// TIA Portal project "LAB3Simu" (V18)

(* hardware
DEVICE "S7-1500/ET200MP station_1"  S7-1500 station
   slot 0: "Rail_0"  Rack  6ES7 590-1***0-0AA0
   slot 1: "PLC_1"  CPU 1511-1 PN  6ES7 511-1AK00-0AB0  V1.8
      slot 3: "CPU display_1"  6ES7591-1AA00-0AA0
      slot 32768: "PROFINET interface_1"  X1
         slot 32769: "Port_1"  X1 P1
         slot 32770: "Port_2"  X1 P2
   slot 2: "CM 1542-5_1"  CM 1542-5  6GK7 542-5DX00-0XE0  V1.0
   slot 3: "DI 16x24VDC HF_1"  DI 16x24VDC HF  6ES7 521-1BH00-0AB0  V1.0
   slot 4: "DQ 16x24VDC/0.5A ST_1"  DQ 16x24VDC/0.5A ST  6ES7 522-1BH00-0AB0  V1.0
   slot 5: "AI 8xU/I/RTD/TC ST_1"  AI 8xU/I/RTD/TC ST  6ES7 531-7KF00-0AB0  V1.0
   slot 6: "AQ 4xU/I ST_1"  AQ 4xU/I ST  6ES7 532-5HD00-0AB0  V1.0
DEVICE "HMI_1"  KP700 Comfort
   slot 0: "HMI_1"  KP700 Comfort  6AV2 124-1GC01-0AX0  17.0.0.0
   slot 1: "HMI_RT_1"  KP700 Comfort  6AV2 124-1GC01-0AX0  17.0.0.0
   slot 5: "HMI_1.IE_CP_1"  PROFINET Interface  17.0.0.0
      slot 1: "PROFINET Interface_1"  PROFINET Interface
         slot 1: "Port_1"  Port
         slot 2: "Port_2"  Port
   slot 7: "HMI_1.MPI/DP_CP_1"  MPI/DP Interface  17.0.0.0
*)

// ===== PLC "PLC_1"  CPU 1511-1 PN =====

VAR_GLOBAL   // PLC tag table "Default tag table"
   "Btn_Ciclo_INIT" AT %M0.0 : Bool;
   "Btn_Ciclo_Cont" AT %M0.1 : Bool;
   "Btn_Parada" AT %M0.2 : Bool;
   "Btn_Emergencia" AT %M0.3 : Bool;
   "Sens_PP" AT %M0.4 : Bool;
   "Sens_PC" AT %M0.5 : Bool;
   "Sens_SM" AT %M0.6 : Bool;
   "A0" AT %M0.7 : Bool;
   "B0" AT %M1.0 : Bool;
   "C0" AT %M1.1 : Bool;
   "D0" AT %M1.2 : Bool;
   "E0" AT %M1.3 : Bool;
   "F0" AT %M1.4 : Bool;
   "A1" AT %M1.5 : Bool;
   "B1" AT %M1.6 : Bool;
   "C1" AT %M1.7 : Bool;
   "D1" AT %M2.0 : Bool;
   "E1" AT %M2.1 : Bool;
   "F1" AT %M2.2 : Bool;
   "Cil_A_+" AT %M2.3 : Bool;
   "Cil_A_-" AT %M2.4 : Bool;
   "Cil_B_Out" AT %M2.5 : Bool;
   "Cil_C_Out" AT %M2.6 : Bool;
   "Cil_D_Out" AT %M2.7 : Bool;
   "Cil_E_+" AT %M3.0 : Bool;
   "Cil_E_-" AT %M3.1 : Bool;
   "Cil_F_+" AT %M3.2 : Bool;
   "Cil_F_-" AT %M3.3 : Bool;
   "Alarma_Stock" AT %M3.4 : Bool;
   "Marca_D_OK" AT %M3.5 : Bool;
   "reset" AT %M3.6 : Bool;
   "start" AT %M3.7 : Bool;
   "stop" AT %M4.0 : Bool;
   "PE" AT %M4.1 : Bool;
   "ALM_start" AT %M4.2 : Bool;
   "ALM_stop" AT %M4.3 : Bool;
   "ALM_em" AT %M4.4 : Bool;
   "block_start" AT %M4.5 : Bool;
   "Alarma_pp" AT %M4.6 : Bool;
   "Alarma_pc" AT %M4.7 : Bool;
   "Marca_start" AT %M5.0 : Bool;
END_VAR

DATA_BLOCK "GRAFCET_DB"   // DB2
{ S7_Optimized_Access := 'TRUE' }
VERSION : 0.1
// stored: InstanceOfName GRAFCET
"GRAFCET"
BEGIN
END_DATA_BLOCK

DATA_BLOCK "FUB_DB"   // DB3
{ S7_Optimized_Access := 'TRUE' }
VERSION : 0.1
// stored: InstanceOfName FUB
"FUB"
BEGIN
END_DATA_BLOCK

DATA_BLOCK "AWL_DB"   // DB4
{ S7_Optimized_Access := 'TRUE' }
VERSION : 0.1
// stored: InstanceOfName AWL
"AWL"
BEGIN
END_DATA_BLOCK

// folder: System blocks/Program resources

DATA_BLOCK "IEC_Timer_0_DB"   // DB1
{ S7_Optimized_Access := 'TRUE' }
AUTHOR : Simatic
FAMILY : IEC
NAME : IEC_TMR
VERSION : 1.0
// stored: InstanceOfName IEC_TIMER
"IEC_TIMER"
BEGIN
END_DATA_BLOCK

// folder: (top level)

FUNCTION_BLOCK "GRAFCET"   // FB1, GRAPH_PLUS
{ S7_Optimized_Access := 'TRUE' }
VERSION : 0.1
   VAR_INPUT
      OFF_SQ : Bool := false;   // Turn sequence off
      INIT_SQ : Bool := false;   // Set sequence to initial state
      ACK_EF : Bool := false;   // Acknowledge all errors and faults
      S_PREV : Bool := false;   // Output previous step in parameter S_NO
      S_NEXT : Bool := false;   // Indicate next step in parameter S_NO
      SW_AUTO : Bool := false;   // Automatic mode
      SW_TAP : Bool := false;   // Semiautomatic/switch with transition
      SW_TOP : Bool := false;   // Semiautomatic/ignore transition
      SW_MAN : Bool := false;   // Manual mode
      S_SEL : Int := 0;   // Select step to be output to S_NO
      S_ON : Bool := false;   // Activate step indicated in S_NO
      S_OFF : Bool := false;   // Disable step indicated in S_NO
      T_PUSH : Bool := false;   // Enable transition to switch in semi automatic mode
   END_VAR
   VAR_OUTPUT
      S_NO : Int := 0;   // Step number
      S_MORE : Bool := false;   // More steps are available and can be shown in S_NO
      S_ACTIVE : Bool := false;   // Step indicated in S_NO is active
      ERR_FLT : Bool := false;   // Interlock or supervision group error
      AUTO_ON : Bool := false;   // Automatic mode is active
      TAP_ON : Bool := false;   // Semiautomatic mode/step with transition enabled
      TOP_ON : Bool := false;   // Semiautomatic mode/ignore transition enabled
      MAN_ON : Bool := false;   // Manual mode is active
   END_VAR
   VAR
      HMI_INFO : Array[0..8] of UInt;
      IF_PAR : G7_IfParPlus_V2;
      RT_DATA : G7_RTDataPlus_V2;   // Internal data area
      Trans1 : G7_TransitionPlus_V2;   // Transition structure
      Trans2 : G7_TransitionPlus_V2;   // Transition structure
      Trans3 : G7_TransitionPlus_V2;   // Transition structure
      Trans4 : G7_TransitionPlus_V2;   // Transition structure
      Trans5 : G7_TransitionPlus_V2;   // Transition structure
      Trans6 : G7_TransitionPlus_V2;   // Transition structure
      Trans7 : G7_TransitionPlus_V2;   // Transition structure
      Trans8 : G7_TransitionPlus_V2;   // Transition structure
      Trans9 : G7_TransitionPlus_V2;   // Transition structure
      Trans10 : G7_TransitionPlus_V2;   // Transition structure
      Trans11 : G7_TransitionPlus_V2;   // Transition structure
      Trans12 : G7_TransitionPlus_V2;   // Transition structure
      Trans13 : G7_TransitionPlus_V2;   // Transition structure
      Trans14 : G7_TransitionPlus_V2;   // Transition structure
      Trans15 : G7_TransitionPlus_V2;   // Transition structure
      Trans16 : G7_TransitionPlus_V2;   // Transition structure
      Trans17 : G7_TransitionPlus_V2;   // Transition structure
      Trans18 : G7_TransitionPlus_V2;   // Transition structure
      Trans19 : G7_TransitionPlus_V2;   // Transition structure
      Trans20 : G7_TransitionPlus_V2;   // Transition structure
      Trans21 : G7_TransitionPlus_V2;   // Transition structure
      Trans22 : G7_TransitionPlus_V2;   // Transition structure
      Trans23 : G7_TransitionPlus_V2;   // Transition structure
      "Reset/Reposo" : G7_StepPlus_V2;   // Step structure
      "A+" : G7_StepPlus_V2;   // Step structure
      "A-" : G7_StepPlus_V2;   // Step structure
      "B+" : G7_StepPlus_V2;   // Step structure
      "C+" : G7_StepPlus_V2;   // Step structure
      "B-" : G7_StepPlus_V2;   // Step structure
      "D sale" : G7_StepPlus_V2;   // Step structure
      "D-" : G7_StepPlus_V2;   // Step structure
      "C-" : G7_StepPlus_V2;   // Step structure
      "E+,F+" : G7_StepPlus_V2;   // Step structure
      "E-,F-" : G7_StepPlus_V2;   // Step structure
      "A++" : G7_StepPlus_V2;   // Step structure
      "A--" : G7_StepPlus_V2;   // Step structure
      "B++" : G7_StepPlus_V2;   // Step structure
      "C++" : G7_StepPlus_V2;   // Step structure
      "B--" : G7_StepPlus_V2;   // Step structure
      D_out : G7_StepPlus_V2;   // Step structure
      "D++" : G7_StepPlus_V2;   // Step structure
      "D--" : G7_StepPlus_V2;   // Step structure
      "E,F++" : G7_StepPlus_V2;   // Step structure
      "E,F--" : G7_StepPlus_V2;   // Step structure
      "Cilindros -" : G7_StepPlus_V2;   // Step structure
      SINI : Array[0..1] of USInt;
      LSTT : Array[0..22] of USInt;
      ATAJ : Array[0..22] of USInt;
      ATAB : Array[0..22] of USInt;
      PSTT : Array[0..22] of USInt;
      NSTT : Array[0..22] of USInt;
      ASSJ : Array[0..21] of USInt;
      ASSB : Array[0..21] of USInt;
      PTTS : Array[0..21] of USInt;
      NTTS : Array[0..21] of USInt;
      SW_SQTS : Array[0..21] of USInt;
      SWITCH : Array[0..1] of USInt;
      TVX : Array[0..3] of USInt;
      TTX : Array[0..3] of USInt;
      TSX : Array[0..1] of USInt;
      S00X : Array[0..1] of USInt;
      SOFFX : Array[0..1] of USInt;
      SONX : Array[0..1] of USInt;
      SAX : Array[0..1] of USInt;
      SERRX : Array[0..22] of USInt;
      SMX : Array[0..22] of USInt;
      S0X : Array[0..22] of USInt;
      S1X : Array[0..22] of USInt;
      IL_ALARM_INST : Program_Alarm;
      SUP_ALARM_INST : Program_Alarm;
      STEP_TIME_ALARM_INST : Program_Alarm;
      IEC_TIMER_INST : IEC_TIMER;
      TRANSACTION_FLAG : Bool := false;
   END_VAR
   // SINI[0] := 2;
   // LSTT[0] := 255;
   // LSTT[1] := 255;
   // LSTT[2] := 255;
   // LSTT[3] := 255;
   // LSTT[4] := 255;
   // LSTT[5] := 255;
   // LSTT[6] := 255;
   // LSTT[7] := 255;
   // LSTT[8] := 255;
   // LSTT[9] := 255;
   // LSTT[10] := 255;
   // LSTT[11] := 255;
   // LSTT[12] := 255;
   // LSTT[13] := 255;
   // LSTT[14] := 255;
   // LSTT[15] := 255;
   // LSTT[16] := 255;
   // LSTT[17] := 255;
   // LSTT[18] := 255;
   // LSTT[19] := 255;
   // LSTT[20] := 255;
   // ATAJ[1] := 1;
   // ATAJ[2] := 2;
   // ATAJ[3] := 3;
   // ATAJ[4] := 4;
   // ATAJ[5] := 5;
   // ATAJ[6] := 6;
   // ATAJ[7] := 7;
   // ATAJ[8] := 8;
   // ATAJ[9] := 9;
   // ATAJ[10] := 10;
   // ATAJ[11] := 11;
   // ATAJ[12] := 12;
   // ATAJ[13] := 13;
   // ATAJ[14] := 14;
   // ATAJ[15] := 15;
   // ATAJ[16] := 16;
   // ATAJ[17] := 17;
   // ATAJ[18] := 18;
   // ATAJ[19] := 19;
   // ATAJ[20] := 20;
   // ATAJ[21] := 21;
   // ATAB[0] := 11;
   // ATAB[1] := 1;
   // ATAB[2] := 2;
   // ATAB[3] := 3;
   // ATAB[4] := 4;
   // ATAB[5] := 5;
   // ATAB[6] := 6;
   // ATAB[7] := 7;
   // ATAB[8] := 8;
   // ATAB[9] := 9;
   // ATAB[10] := 10;
   // ATAB[12] := 12;
   // ATAB[13] := 13;
   // ATAB[14] := 14;
   // ATAB[15] := 15;
   // ATAB[16] := 16;
   // ATAB[17] := 17;
   // ATAB[18] := 18;
   // ATAB[19] := 19;
   // ATAB[20] := 20;
   // ATAB[21] := 21;
   // PSTT[1] := 1;
   // PSTT[2] := 2;
   // PSTT[3] := 3;
   // PSTT[4] := 4;
   // PSTT[5] := 5;
   // PSTT[6] := 6;
   // PSTT[7] := 7;
   // PSTT[8] := 8;
   // PSTT[9] := 9;
   // PSTT[10] := 10;
   // PSTT[12] := 11;
   // PSTT[13] := 12;
   // PSTT[14] := 13;
   // PSTT[15] := 14;
   // PSTT[16] := 15;
   // PSTT[17] := 16;
   // PSTT[18] := 17;
   // PSTT[19] := 18;
   // PSTT[20] := 19;
   // PSTT[21] := 20;
   // NSTT[0] := 1;
   // NSTT[1] := 2;
   // NSTT[2] := 3;
   // NSTT[3] := 4;
   // NSTT[4] := 5;
   // NSTT[5] := 6;
   // NSTT[6] := 7;
   // NSTT[7] := 8;
   // NSTT[8] := 9;
   // NSTT[9] := 10;
   // NSTT[10] := 255;
   // NSTT[11] := 11;
   // NSTT[12] := 12;
   // NSTT[13] := 13;
   // NSTT[14] := 14;
   // NSTT[15] := 15;
   // NSTT[16] := 16;
   // NSTT[17] := 17;
   // NSTT[18] := 18;
   // NSTT[19] := 19;
   // NSTT[20] := 20;
   // ASSJ[1] := 1;
   // ASSJ[2] := 2;
   // ASSJ[3] := 3;
   // ASSJ[4] := 4;
   // ASSJ[5] := 5;
   // ASSJ[6] := 6;
   // ASSJ[7] := 7;
   // ASSJ[8] := 8;
   // ASSJ[9] := 9;
   // ASSJ[10] := 10;
   // ASSJ[11] := 11;
   // ASSJ[12] := 12;
   // ASSJ[13] := 13;
   // ASSJ[14] := 14;
   // ASSJ[15] := 15;
   // ASSJ[16] := 16;
   // ASSJ[17] := 17;
   // ASSJ[18] := 18;
   // ASSJ[19] := 19;
   // ASSJ[20] := 20;
   // ASSB[1] := 1;
   // ASSB[2] := 2;
   // ASSB[3] := 3;
   // ASSB[4] := 4;
   // ASSB[5] := 5;
   // ASSB[6] := 6;
   // ASSB[7] := 7;
   // ASSB[8] := 8;
   // ASSB[9] := 9;
   // ASSB[10] := 10;
   // ASSB[11] := 11;
   // ASSB[12] := 12;
   // ASSB[13] := 13;
   // ASSB[14] := 14;
   // ASSB[15] := 15;
   // ASSB[16] := 16;
   // ASSB[17] := 17;
   // ASSB[18] := 18;
   // ASSB[19] := 19;
   // ASSB[20] := 20;
   // PTTS[0] := 255;
   // PTTS[2] := 1;
   // PTTS[3] := 2;
   // PTTS[4] := 3;
   // PTTS[5] := 4;
   // PTTS[6] := 5;
   // PTTS[7] := 6;
   // PTTS[8] := 7;
   // PTTS[9] := 8;
   // PTTS[10] := 9;
   // PTTS[11] := 11;
   // PTTS[12] := 12;
   // PTTS[13] := 13;
   // PTTS[14] := 14;
   // PTTS[15] := 15;
   // PTTS[16] := 16;
   // PTTS[17] := 17;
   // PTTS[18] := 18;
   // PTTS[19] := 19;
   // PTTS[20] := 20;
   // NTTS[1] := 1;
   // NTTS[2] := 2;
   // NTTS[3] := 3;
   // NTTS[4] := 4;
   // NTTS[5] := 5;
   // NTTS[6] := 6;
   // NTTS[7] := 7;
   // NTTS[8] := 8;
   // NTTS[9] := 9;
   // NTTS[10] := 10;
   // NTTS[11] := 12;
   // NTTS[12] := 13;
   // NTTS[13] := 14;
   // NTTS[14] := 15;
   // NTTS[15] := 16;
   // NTTS[16] := 17;
   // NTTS[17] := 18;
   // NTTS[18] := 19;
   // NTTS[19] := 20;
   // NTTS[20] := 21;
   // SW_SQTS[1] := 1;
   // SW_SQTS[2] := 1;
   // SW_SQTS[3] := 1;
   // SW_SQTS[4] := 1;
   // SW_SQTS[5] := 1;
   // SW_SQTS[6] := 1;
   // SW_SQTS[7] := 1;
   // SW_SQTS[8] := 1;
   // SW_SQTS[9] := 1;
   // SW_SQTS[10] := 1;
   // SW_SQTS[11] := 2;
   // SW_SQTS[12] := 2;
   // SW_SQTS[13] := 2;
   // SW_SQTS[14] := 2;
   // SW_SQTS[15] := 2;
   // SW_SQTS[16] := 2;
   // SW_SQTS[17] := 2;
   // SW_SQTS[18] := 2;
   // SW_SQTS[19] := 2;
   // SW_SQTS[20] := 2;
   // TVX[0] := 16#1;
   // TTX[0] := 16#1;
   // TSX[0] := 16#1;
   // S00X[0] := 16#1;
   // SOFFX[0] := 16#1;
   // SONX[0] := 16#1;
   // SAX[0] := 16#1;
   // SERRX[0] := 16#1;
   // SMX[0] := 16#1;
   // S0X[0] := 16#1;
   // S1X[0] := 16#1;
   // LSTT[22] := 255;
   // ATAJ[22] := 22;
   // ATAB[22] := 22;
   // PSTT[0] := 21;
   // PSTT[11] := 21;
   // NSTT[22] := 21;
   // ASSJ[21] := 21;
   // ASSB[21] := 21;
   // PTTS[21] := 22;
   // NTTS[0] := 22;
BEGIN
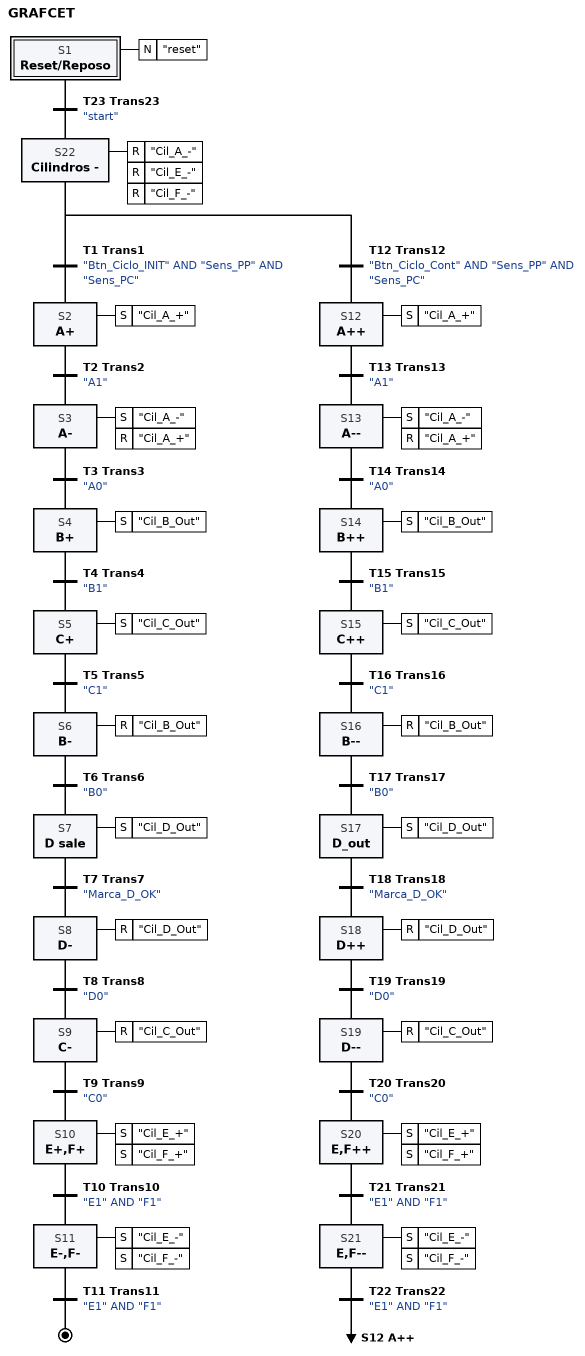
   // sequencer 1
   INITIAL_STEP "Reset/Reposo":   // S1, max time T#10S, warning time T#7S
              N    "reset"
   END_STEP
   TRANSITION Trans23 FROM "Reset/Reposo" TO "Cilindros -"   // T23
      := "start";
   END_TRANSITION
   STEP "A+":   // S2, max time T#10S, warning time T#7S
              S    "Cil_A_+"
   END_STEP
   TRANSITION Trans2 FROM "A+" TO "A-"   // T2
      := "A1";
   END_TRANSITION
   STEP "A-":   // S3, max time T#10S, warning time T#7S
              S    "Cil_A_-"
              R    "Cil_A_+"
   END_STEP
   TRANSITION Trans3 FROM "A-" TO "B+"   // T3
      := "A0";
   END_TRANSITION
   STEP "B+":   // S4, max time T#10S, warning time T#7S
              S    "Cil_B_Out"
   END_STEP
   TRANSITION Trans4 FROM "B+" TO "C+"   // T4
      := "B1";
   END_TRANSITION
   STEP "C+":   // S5, max time T#10S, warning time T#7S
              S    "Cil_C_Out"
   END_STEP
   TRANSITION Trans5 FROM "C+" TO "B-"   // T5
      := "C1";
   END_TRANSITION
   STEP "B-":   // S6, max time T#10S, warning time T#7S
              R    "Cil_B_Out"
   END_STEP
   TRANSITION Trans6 FROM "B-" TO "D sale"   // T6
      := "B0";
   END_TRANSITION
   STEP "D sale":   // S7, max time T#10S, warning time T#7S
              S    "Cil_D_Out"
   END_STEP
   TRANSITION Trans7 FROM "D sale" TO "D-"   // T7
      := "Marca_D_OK";
   END_TRANSITION
   STEP "D-":   // S8, max time T#10S, warning time T#7S
              R    "Cil_D_Out"
   END_STEP
   TRANSITION Trans8 FROM "D-" TO "C-"   // T8
      := "D0";
   END_TRANSITION
   STEP "C-":   // S9, max time T#10S, warning time T#7S
              R    "Cil_C_Out"
   END_STEP
   TRANSITION Trans9 FROM "C-" TO "E+,F+"   // T9
      := "C0";
   END_TRANSITION
   STEP "E+,F+":   // S10, max time T#10S, warning time T#7S
              S    "Cil_E_+"
              S    "Cil_F_+"
   END_STEP
   TRANSITION Trans10 FROM "E+,F+" TO "E-,F-"   // T10
      := "E1" AND "F1";
   END_TRANSITION
   STEP "E-,F-":   // S11, max time T#10S, warning time T#7S
              S    "Cil_E_-"
              S    "Cil_F_-"
   END_STEP
   TRANSITION Trans11 FROM "E-,F-" TO END   // T11
      := "E1" AND "F1";
   END_TRANSITION
   STEP "A++":   // S12, max time T#10S, warning time T#7S
              S    "Cil_A_+"
   END_STEP
   TRANSITION Trans13 FROM "A++" TO "A--"   // T13
      := "A1";
   END_TRANSITION
   STEP "A--":   // S13, max time T#10S, warning time T#7S
              S    "Cil_A_-"
              R    "Cil_A_+"
   END_STEP
   TRANSITION Trans14 FROM "A--" TO "B++"   // T14
      := "A0";
   END_TRANSITION
   STEP "B++":   // S14, max time T#10S, warning time T#7S
              S    "Cil_B_Out"
   END_STEP
   TRANSITION Trans15 FROM "B++" TO "C++"   // T15
      := "B1";
   END_TRANSITION
   STEP "C++":   // S15, max time T#10S, warning time T#7S
              S    "Cil_C_Out"
   END_STEP
   TRANSITION Trans16 FROM "C++" TO "B--"   // T16
      := "C1";
   END_TRANSITION
   STEP "B--":   // S16, max time T#10S, warning time T#7S
              R    "Cil_B_Out"
   END_STEP
   TRANSITION Trans17 FROM "B--" TO D_out   // T17
      := "B0";
   END_TRANSITION
   STEP D_out:   // S17, max time T#10S, warning time T#7S
              S    "Cil_D_Out"
   END_STEP
   TRANSITION Trans18 FROM D_out TO "D++"   // T18
      := "Marca_D_OK";
   END_TRANSITION
   STEP "D++":   // S18, max time T#10S, warning time T#7S
              R    "Cil_D_Out"
   END_STEP
   TRANSITION Trans19 FROM "D++" TO "D--"   // T19
      := "D0";
   END_TRANSITION
   STEP "D--":   // S19, max time T#10S, warning time T#7S
              R    "Cil_C_Out"
   END_STEP
   TRANSITION Trans20 FROM "D--" TO "E,F++"   // T20
      := "C0";
   END_TRANSITION
   STEP "E,F++":   // S20, max time T#10S, warning time T#7S
              S    "Cil_E_+"
              S    "Cil_F_+"
   END_STEP
   TRANSITION Trans21 FROM "E,F++" TO "E,F--"   // T21
      := "E1" AND "F1";
   END_TRANSITION
   STEP "E,F--":   // S21, max time T#10S, warning time T#7S
              S    "Cil_E_-"
              S    "Cil_F_-"
   END_STEP
   TRANSITION Trans22 FROM "E,F--" TO "A++"   // T22, jump
      := "E1" AND "F1";
   END_TRANSITION
   STEP "Cilindros -":   // S22, max time T#10S, warning time T#7S
              R    "Cil_A_-"
              R    "Cil_E_-"
              R    "Cil_F_-"
   END_STEP
   TRANSITION Trans1 FROM "Cilindros -" TO "A+"   // T1
      := "Btn_Ciclo_INIT" AND "Sens_PP" AND "Sens_PC";
   END_TRANSITION
   TRANSITION Trans12 FROM "Cilindros -" TO "A++"   // T12
      := "Btn_Ciclo_Cont" AND "Sens_PP" AND "Sens_PC";
   END_TRANSITION
END_FUNCTION_BLOCK

FUNCTION_BLOCK "AWL"   // FB2, STL
{ S7_Optimized_Access := 'TRUE' }
VERSION : 0.1
BEGIN

REGION Network 1
         A     "reset";

         R     "Cil_A_+";
         S     "Cil_A_-";
         R     "Cil_E_+";
         S     "Cil_E_-";
         R     "Cil_F_+";
         S     "Cil_F_-";

         R     "Cil_B_Out";
         R     "Cil_C_Out";
         R     "Cil_D_Out";

         R     "Alarma_Stock";
         R     "Alarma_pc";
         S     "ALM_em";
         R     "Alarma_pp";
         R     "ALM_start";
         R     "ALM_stop";
END_REGION
END_FUNCTION_BLOCK

FUNCTION_BLOCK "FUB"   // FB3, FBD
{ S7_Optimized_Access := 'TRUE' }
VERSION : 0.1
BEGIN

REGION Network 1
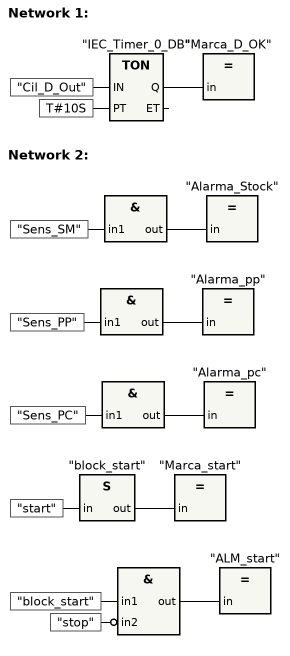
   "IEC_Timer_0_DB".TON(IN := "Cil_D_Out", PT := T#10S);
   "Marca_D_OK" := "IEC_Timer_0_DB".Q;
END_REGION

REGION Network 2
   "Alarma_Stock" := "Sens_SM";
   "Alarma_pp" := "Sens_PP";
   "Alarma_pc" := "Sens_PC";
   IF "start" THEN "block_start" := TRUE; END_IF;
   "Marca_start" := "start";
   "ALM_start" := "block_start" AND NOT "stop";
END_REGION
END_FUNCTION_BLOCK

ORGANIZATION_BLOCK "Main"   // OB1, LAD, ProgramCycle
TITLE = "Main Program Sweep (Cycle)"
{ S7_Optimized_Access := 'TRUE' }
VERSION : 0.1
   VAR_INPUT
      Initial_Call : Bool;   // Initial call of this OB
      Remanence : Bool;   // =True, if remanent data are available
   END_VAR
BEGIN

REGION Network 1
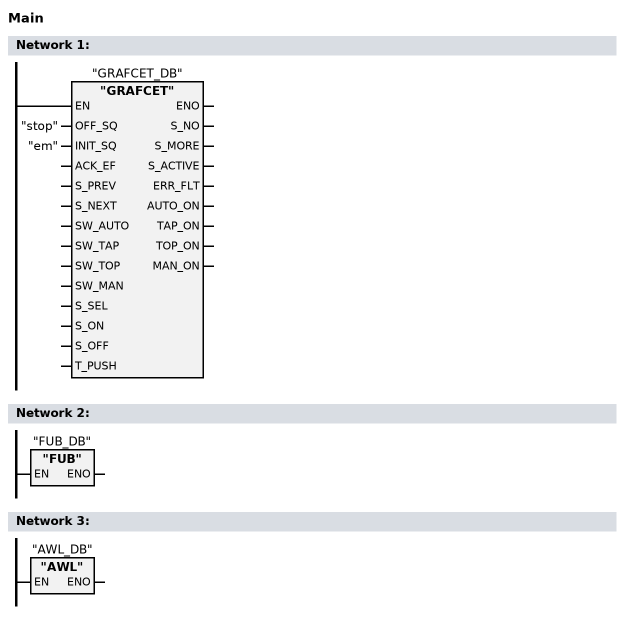
   RUNG wire#powerrail
      "GRAFCET_DB"(OFF_SQ := "stop", INIT_SQ := "em", ACK_EF :=, S_PREV :=, S_NEXT :=, SW_AUTO :=, SW_TAP :=, SW_TOP :=, SW_MAN :=, S_SEL :=, S_ON :=, S_OFF :=, T_PUSH :=, S_NO =>, S_MORE =>, S_ACTIVE =>, ERR_FLT =>, AUTO_ON =>, TAP_ON =>, TOP_ON =>, MAN_ON =>)
   END_RUNG
   // the same network as SCL:
   "GRAFCET_DB"(OFF_SQ := "stop", INIT_SQ := "em");   // "GRAFCET"
END_REGION

REGION Network 2
   RUNG wire#powerrail
      "FUB_DB"()
   END_RUNG
   // the same network as SCL:
   "FUB_DB"();   // "FUB"
END_REGION

REGION Network 3
   RUNG wire#powerrail
      "AWL_DB"()
   END_RUNG
   // the same network as SCL:
   "AWL_DB"();   // "AWL"
END_REGION
END_ORGANIZATION_BLOCK

(* ===== HMI "HMI_RT_1" =====
system functions are stored by id; their names below are inferred from use
connection "HMI_Connection_1": ETHERNET, S7_1500_OMS

HMI tags "Default tag table"
   "Alarma_Stock" : Bool = PLC Alarma_Stock AT %M3.4, 1 s
   "Btn_Ciclo_Unico" : Bool = PLC Btn_Ciclo_INIT AT %M0.0, 1 s
   "Btn_Ciclo_Cont" : Bool = PLC Btn_Ciclo_Cont AT %M0.1, 1 s
   "indi_start" : Bool = PLC ALM_start AT %M4.2, 1 s
   "indi_stop" : Bool = PLC ALM_stop AT %M4.3, 1 s
   "indi_em" : Bool = PLC ALM_em AT %M4.4, 1 s
   "A1" : Bool = PLC A1 AT %M1.5, 1 s
   "B1" : Bool = PLC B1 AT %M1.6, 1 s
   "C1" : Bool = PLC C1 AT %M1.7, 1 s
   "D1" : Bool = PLC D1 AT %M2.0, 1 s
   "E1" : Bool = PLC E1 AT %M2.1, 1 s
   "F1" : Bool = PLC F1 AT %M2.2, 1 s
   "Alarma_pp" : Bool = PLC Alarma_pp AT %M4.6, 1 s
   "Alarma_pc" : Bool = PLC Alarma_pc AT %M4.7, 1 s
   "start" : Bool = PLC start AT %M3.7, 1 s

screen "Screen_1" 800x480
   Button "Button_1" at 1,12 size 96x32; TextOff 'Start'
      on Press: SetBit("start")
   Button "Button_2" at 1,67 size 96x32; TextOff 'Stop'
   Button "Button_3" at 1,124 size 96x32; TextOff 'Emergencia'
   Circle "Circle_1" at 120,89 size 48x48
      Appearance <- "indi_start"
   Circle "Circle_2" at 180,89 size 48x48
      Appearance <- "indi_stop"
   Circle "Circle_3" at 244,89 size 48x48
      Appearance <- "indi_em"
   TextField "Text field_1" at 134,2 size 60x21; Text 'Prueba'
   TextField "Text field_2" at 242,3 size 41x21; Text 'Ciclo'
   TextField "Text field_4" at 127,104 size 31x15; Text 'Start'
   TextField "Text field_5" at 191,103 size 28x15; Text 'Stop'
   TextField "Text field_6" at 258,104 size 19x15; Text 'Em'
   Switch "Switch_1" at 130,24 size 64x32; CaptionText 'Switch'; TextOff 'OFF'; TextOn 'ON'
      on SwitchOn: SetBit("Btn_Ciclo_Unico")
      on SwitchOff: ResetBit("Btn_Ciclo_Unico")
   Switch "Switch_2" at 232,23 size 64x32; CaptionText 'Switch'; TextOff 'OFF'; TextOn 'ON'
      on SwitchOn: SetBit("Btn_Ciclo_Cont")
      on SwitchOff: ResetBit("Btn_Ciclo_Cont")
   GraphicView "Graphic view_1" at 120,159 size 48x29; Picture "Graphic_10"
      Visibility <- "A1"
   GraphicView "Graphic view_2" at 120,210 size 48x29; Picture "Graphic_10"
      Visibility <- "D1"
   GraphicView "Graphic view_3" at 189,158 size 48x29; Picture "Graphic_10"
      Visibility <- "B1"
   GraphicView "Graphic view_4" at 189,210 size 48x29; Picture "Graphic_10"
      Visibility <- "E1"
   GraphicView "Graphic view_5" at 252,158 size 48x29; Picture "Graphic_10"
      Visibility <- "C1"
   GraphicView "Graphic view_6" at 252,210 size 48x29; Picture "Graphic_10"
      Visibility <- "F1"
   GraphicView "Graphic view_7" at -3,181 size 92x20; Picture "Graphic_11"
      Visibility <- "Alarma_Stock"
   GraphicView "Graphic view_8" at -2,198 size 91x18; Picture "Graphic_12"
      Visibility <- "Alarma_pp"
   GraphicView "Graphic view_9" at -1,215 size 90x18; Picture "Graphic_13"
      Visibility <- "Alarma_pc"
   TextField "Text field_3" at 130,141 size 12x18; Text 'A'
   TextField "Text field_7" at 202,141 size 10x18; Text 'B'
   TextField "Text field_8" at 265,141 size 10x18; Text 'C'
   TextField "Text field_9" at 129,192 size 11x18; Text 'D'
   TextField "Text field_10" at 201,192 size 10x18; Text 'E'
   TextField "Text field_11" at 264,192 size 10x18; Text 'F'
*)